// TIA Portal V16 export
// export: Created 2022-02-28T20:45:45.8704837Z, ExportSetting WithDefaults, DisplayName Totally Integrated Automation Portal, DisplayVersion V16, DisplayName TIA Portal Version Control Interface, DisplayVersion V16, DisplayName TIA Portal Openness, DisplayVersion V16, DisplayName STEP 7 Professional, DisplayVersion V16, DisplayName STEP 7 Safety, DisplayVersion V16, DisplayName WinCC Advanced, DisplayVersion V16
DATA_BLOCK "02_Software-PLC"   // DB2
{ S7_Optimized_Access := 'TRUE' }
VERSION : 0.1
// stored: AutoNumber true, DBAccessibleFromOPCUA true, IsOnlyStoredInLoadMemory false, IsRetainMemResEnabled false, IsWriteProtectedInAS false, MemoryReserve 100
   VAR
      Variables_Generales : Struct
         Multip_Cantiadad_Prod : Real;   // Orden de producción
         Multip_Margen_Prod : Real;   // Margen de error producción
         Multip_Confir_Arranque : Bool;   // Permiso de arranque producción
         Multip_Formato_Trabajo : Int;   // Refencia Cajas
      END_STRUCT;
      Datos_Pentoflex : Struct
         "MPF_Remoto/Local" : Bool;   // Manejo Remoto / Local
         MPF_ModoAuto : Bool;   // Modo Automatico
         MPF_Modo_Manual : Bool;   // Modo Manual
         MPF_Estado_Impresora3 : Bool;   // Estado de la impresora 3
         MPF_Start_Remoto : Bool;   // Start Remoto Pentof
         MPF_Stop_Remoto : Bool;   // Stop Remoto Pentof
         MPF_Reset_Alarmas : Bool;   // Reset Alarma Pentoflex
      END_STRUCT;
      Datos_Pistilos : Struct
         MP_Codigo_Impresion : String;   // codigo de impresión
         MP_Conf_Arranque : Bool;   // Arranque de orden pistilos
         "MP_Remoto/Local" : Bool;   // Manejo Remoto / Local
         MP_ModoAuto : Bool;   // Modo Automatico
         MP_Modo_Manual : Bool;   // Modo Manual
         MP_Estado_Impresora1 : Bool;   // Estado de la impresora 1
         MP_Estado_Impresora2 : Bool;   // Estado de la impresora 2
         MP_Start_Remoto : Bool;   // Start Pistilos Remoto
         MP_Stop_Remoto : Bool;   // Stop Pistilos Remoto
         MP_Cod_Impreso1 : Bool;   // Codigo Impreso
         MP_Reset_Alarmas : Bool;   // Reset Alarmas Pistilos
      END_STRUCT;
   END_VAR
BEGIN
END_DATA_BLOCK
